// Mitsubishi GX Developer project: Пресс 40 (СКО)   PLC: FX3G

PROGRAM MAIN
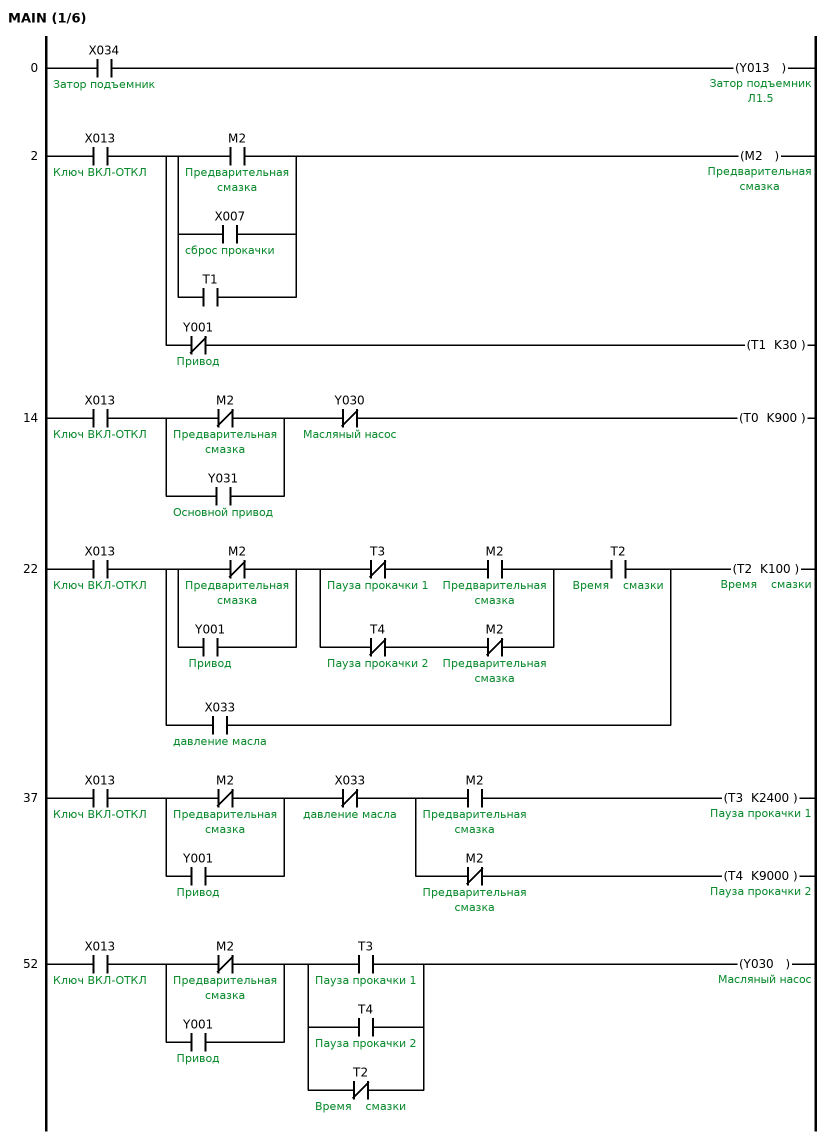
0     LD      X034  ; Затор подъемник
      OUT     Y013  ; Затор подъемник  Л1.5
2     LD      X013  ; Ключ ВКЛ-ОТКЛ
      MPS
      LD      M2  ; Предварительная смазка
      OR      X007  ; сброс прокачки
      OR      T1
      ANB
      OUT     M2  ; Предварительная смазка
      MPP
      ANI     Y001  ; Привод
      OUT     T1 K30
14    LD      X013  ; Ключ ВКЛ-ОТКЛ
      LDI     M2  ; Предварительная смазка
      OR      Y031  ; Основной привод
      ANB
      ANI     Y030  ; Масляный насос
      OUT     T0 K900
22    LD      X013  ; Ключ ВКЛ-ОТКЛ
      LDI     M2  ; Предварительная смазка
      OR      Y001  ; Привод
      LDI     T3  ; Пауза прокачки 1
      AND     M2  ; Предварительная смазка
      LDI     T4  ; Пауза прокачки 2
      ANI     M2  ; Предварительная смазка
      ORB
      ANB
      AND     T2  ; Время    смазки
      OR      X033  ; давление масла
      ANB
      OUT     T2 K100  ; Время    смазки
37    LD      X013  ; Ключ ВКЛ-ОТКЛ
      LDI     M2  ; Предварительная смазка
      OR      Y001  ; Привод
      ANB
      ANI     X033  ; давление масла
      MPS
      AND     M2  ; Предварительная смазка
      OUT     T3 K2400  ; Пауза прокачки 1
      MPP
      ANI     M2  ; Предварительная смазка
      OUT     T4 K9000  ; Пауза прокачки 2
52    LD      X013  ; Ключ ВКЛ-ОТКЛ
      LDI     M2  ; Предварительная смазка
      OR      Y001  ; Привод
      ANB
      LD      T3  ; Пауза прокачки 1
      OR      T4  ; Пауза прокачки 2
      ORI     T2  ; Время    смазки
      ANB
      OUT     Y030  ; Масляный насос
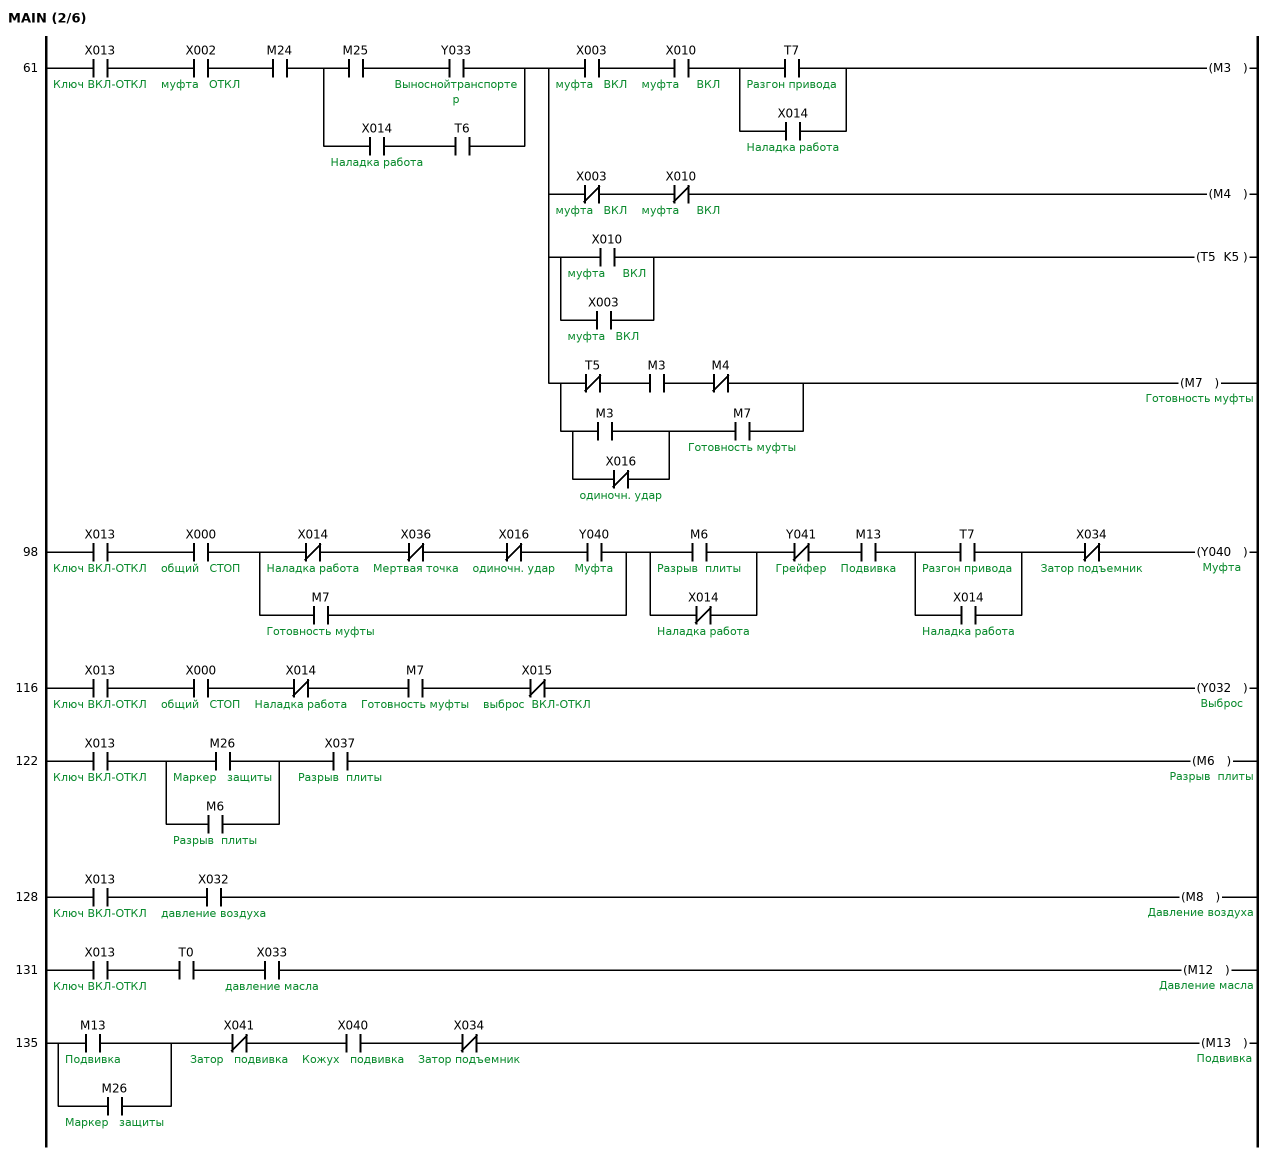
61    LD      X013  ; Ключ ВКЛ-ОТКЛ
      AND     X002  ; муфта   ОТКЛ
      AND     M24
      LD      M25
      AND     Y033  ; Выноснойтранспортер
      LD      X014  ; Наладка работа
      AND     T6
      ORB
      ANB
      MPS
      AND     X003  ; муфта   ВКЛ
      AND     X010  ; муфта     ВКЛ
      LD      T7  ; Разгон привода
      OR      X014  ; Наладка работа
      ANB
      OUT     M3
      MRD
      ANI     X003  ; муфта   ВКЛ
      ANI     X010  ; муфта     ВКЛ
      OUT     M4
      MRD
      LD      X010  ; муфта     ВКЛ
      OR      X003  ; муфта   ВКЛ
      ANB
      OUT     T5 K5
      MPP
      LDI     T5
      AND     M3
      ANI     M4
      LD      M3
      ORI     X016  ; одиночн. удар
      AND     M7  ; Готовность муфты
      ORB
      ANB
      OUT     M7  ; Готовность муфты
98    LD      X013  ; Ключ ВКЛ-ОТКЛ
      AND     X000  ; общий   СТОП
      LDI     X014  ; Наладка работа
      ANI     X036  ; Мертвая точка
      ANI     X016  ; одиночн. удар
      AND     Y040  ; Муфта
      OR      M7  ; Готовность муфты
      ANB
      LD      M6  ; Разрыв  плиты
      ORI     X014  ; Наладка работа
      ANB
      ANI     Y041  ; Грейфер
      AND     M13  ; Подвивка
      LD      T7  ; Разгон привода
      OR      X014  ; Наладка работа
      ANB
      ANI     X034  ; Затор подъемник
      OUT     Y040  ; Муфта
116   LD      X013  ; Ключ ВКЛ-ОТКЛ
      AND     X000  ; общий   СТОП
      ANI     X014  ; Наладка работа
      AND     M7  ; Готовность муфты
      ANI     X015  ; выброс  ВКЛ-ОТКЛ
      OUT     Y032  ; Выброс
122   LD      X013  ; Ключ ВКЛ-ОТКЛ
      LD      M26  ; Маркер   защиты
      OR      M6  ; Разрыв  плиты
      ANB
      AND     X037  ; Разрыв  плиты
      OUT     M6  ; Разрыв  плиты
128   LD      X013  ; Ключ ВКЛ-ОТКЛ
      AND     X032  ; давление воздуха
      OUT     M8  ; Давление воздуха
131   LD      X013  ; Ключ ВКЛ-ОТКЛ
      AND     T0
      AND     X033  ; давление масла
      OUT     M12  ; Давление масла
135   LD      M13  ; Подвивка
      OR      M26  ; Маркер   защиты
      ANI     X041  ; Затор   подвивка
      AND     X040  ; Кожух   подвивка
      ANI     X034  ; Затор подъемник
      OUT     M13  ; Подвивка
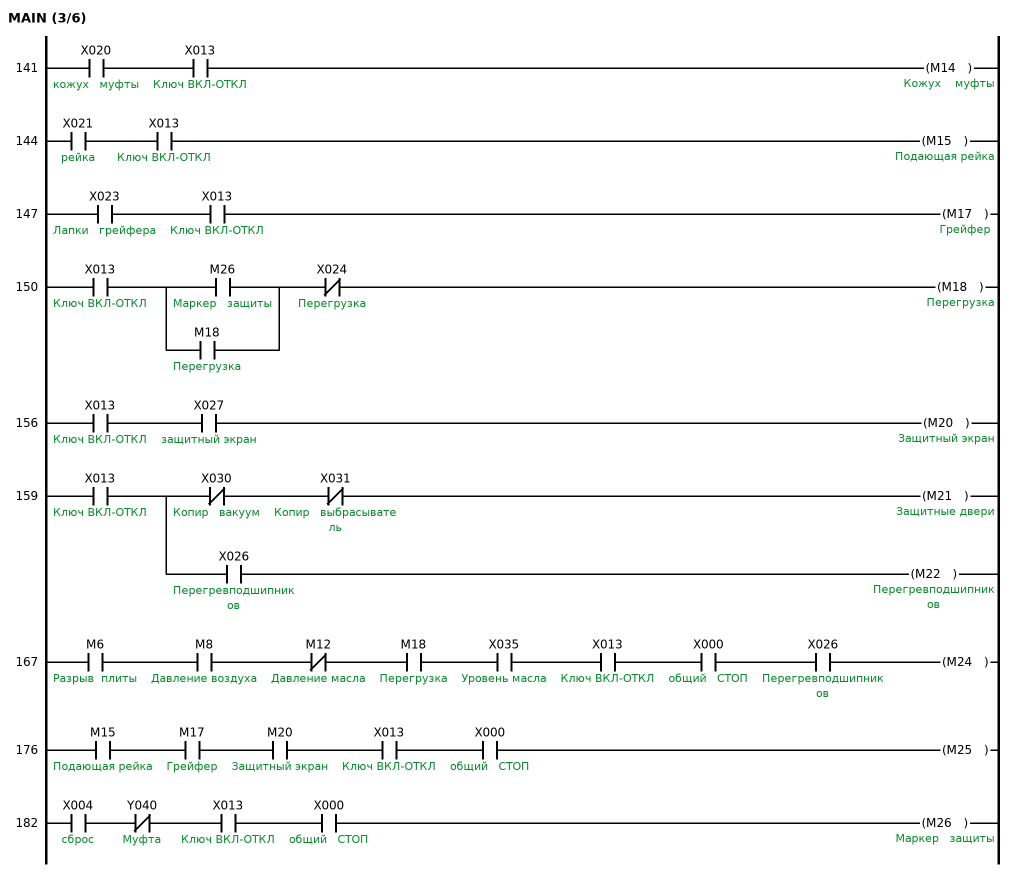
141   LD      X020  ; кожух   муфты
      AND     X013  ; Ключ ВКЛ-ОТКЛ
      OUT     M14  ; Кожух    муфты
144   LD      X021  ; рейка
      AND     X013  ; Ключ ВКЛ-ОТКЛ
      OUT     M15  ; Подающая рейка
147   LD      X023  ; Лапки   грейфера
      AND     X013  ; Ключ ВКЛ-ОТКЛ
      OUT     M17  ; Грейфер
150   LD      X013  ; Ключ ВКЛ-ОТКЛ
      LD      M26  ; Маркер   защиты
      OR      M18  ; Перегрузка
      ANB
      ANI     X024  ; Перегрузка
      OUT     M18  ; Перегрузка
156   LD      X013  ; Ключ ВКЛ-ОТКЛ
      AND     X027  ; защитный экран
      OUT     M20  ; Защитный экран
159   LD      X013  ; Ключ ВКЛ-ОТКЛ
      MPS
      ANI     X030  ; Копир   вакуум
      ANI     X031  ; Копир   выбрасыватель
      OUT     M21  ; Защитные двери
      MPP
      AND     X026  ; Перегревподшипников
      OUT     M22  ; Перегревподшипников
167   LD      M6  ; Разрыв  плиты
      AND     M8  ; Давление воздуха
      ANI     M12  ; Давление масла
      AND     M18  ; Перегрузка
      AND     X035  ; Уровень масла
      AND     X013  ; Ключ ВКЛ-ОТКЛ
      AND     X000  ; общий   СТОП
      AND     X026  ; Перегревподшипников
      OUT     M24
176   LD      M15  ; Подающая рейка
      AND     M17  ; Грейфер
      AND     M20  ; Защитный экран
      AND     X013  ; Ключ ВКЛ-ОТКЛ
      AND     X000  ; общий   СТОП
      OUT     M25
182   LD      X004  ; сброс
      ANI     Y040  ; Муфта
      AND     X013  ; Ключ ВКЛ-ОТКЛ
      AND     X000  ; общий   СТОП
      OUT     M26  ; Маркер   защиты
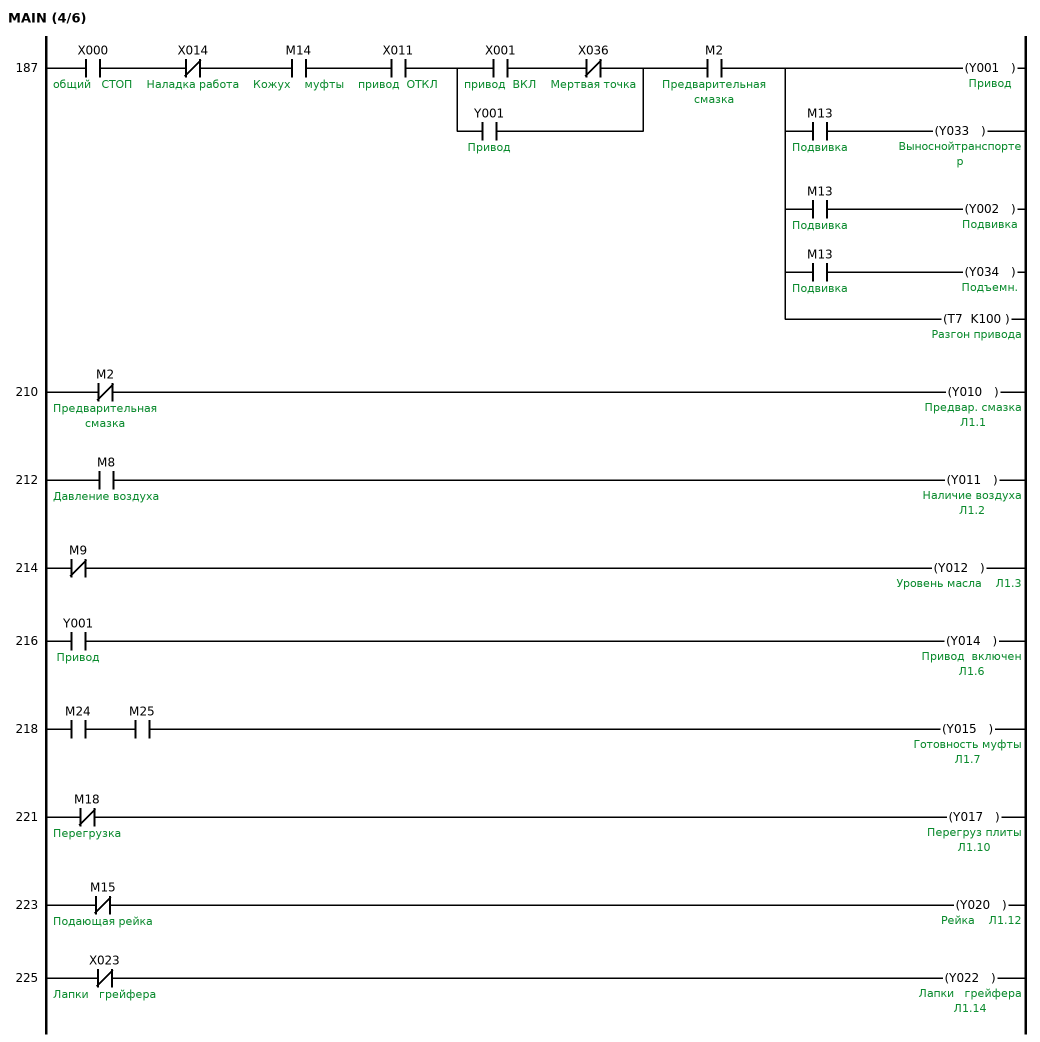
187   LD      X000  ; общий   СТОП
      ANI     X014  ; Наладка работа
      AND     M14  ; Кожух    муфты
      AND     X011  ; привод  ОТКЛ
      LD      X001  ; привод  ВКЛ
      ANI     X036  ; Мертвая точка
      OR      Y001  ; Привод
      ANB
      AND     M2  ; Предварительная смазка
      OUT     Y001  ; Привод
      MPS
      AND     M13  ; Подвивка
      OUT     Y033  ; Выноснойтранспортер
      MRD
      AND     M13  ; Подвивка
      OUT     Y002  ; Подвивка
      MRD
      AND     M13  ; Подвивка
      OUT     Y034  ; Подъемн.
      MPP
      OUT     T7 K100  ; Разгон привода
210   LDI     M2  ; Предварительная смазка
      OUT     Y010  ; Предвар. смазка   Л1.1
212   LD      M8  ; Давление воздуха
      OUT     Y011  ; Наличие воздуха  Л1.2
214   LDI     M9
      OUT     Y012  ; Уровень масла    Л1.3
216   LD      Y001  ; Привод
      OUT     Y014  ; Привод  включен  Л1.6
218   LD      M24
      AND     M25
      OUT     Y015  ; Готовность муфты  Л1.7
221   LDI     M18  ; Перегрузка
      OUT     Y017  ; Перегруз плиты   Л1.10
223   LDI     M15  ; Подающая рейка
      OUT     Y020  ; Рейка    Л1.12
225   LDI     X023  ; Лапки   грейфера
      OUT     Y022  ; Лапки   грейфера  Л1.14
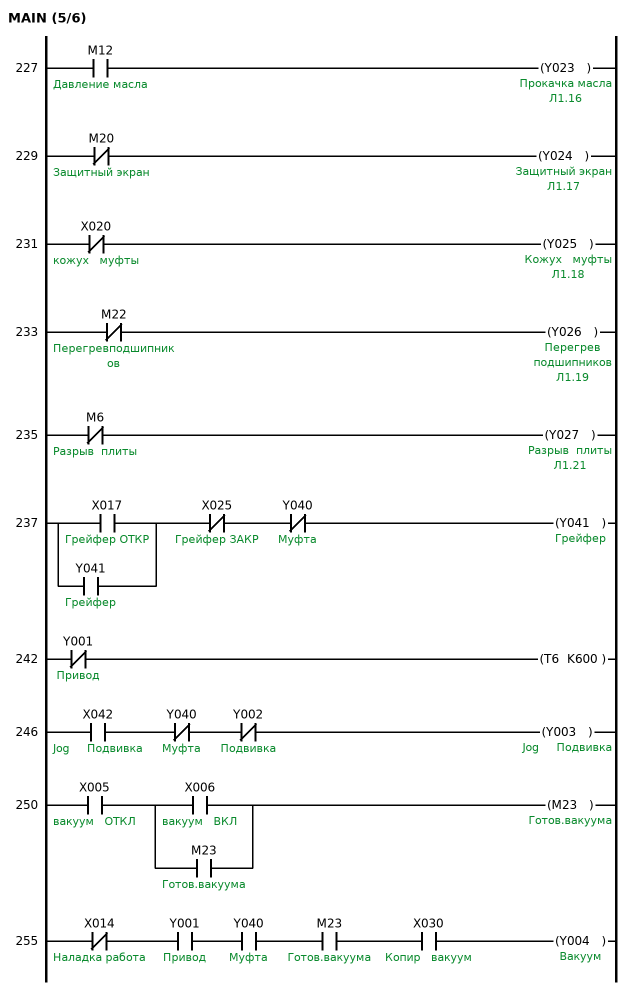
227   LD      M12  ; Давление масла
      OUT     Y023  ; Прокачка масла   Л1.16
229   LDI     M20  ; Защитный экран
      OUT     Y024  ; Защитный экран   Л1.17
231   LDI     X020  ; кожух   муфты
      OUT     Y025  ; Кожух   муфты   Л1.18
233   LDI     M22  ; Перегревподшипников
      OUT     Y026  ; Перегрев подшипников     Л1.19
235   LDI     M6  ; Разрыв  плиты
      OUT     Y027  ; Разрыв  плиты    Л1.21
237   LD      X017  ; Грейфер ОТКР
      OR      Y041  ; Грейфер
      ANI     X025  ; Грейфер ЗАКР
      ANI     Y040  ; Муфта
      OUT     Y041  ; Грейфер
242   LDI     Y001  ; Привод
      OUT     T6 K600
246   LD      X042  ; Jog     Подвивка
      ANI     Y040  ; Муфта
      ANI     Y002  ; Подвивка
      OUT     Y003  ; Jog     Подвивка
250   LD      X005  ; вакуум   ОТКЛ
      LD      X006  ; вакуум   ВКЛ
      OR      M23  ; Готов.вакуума
      ANB
      OUT     M23  ; Готов.вакуума
255   LDI     X014  ; Наладка работа
      AND     Y001  ; Привод
      AND     Y040  ; Муфта
      AND     M23  ; Готов.вакуума
      AND     X030  ; Копир   вакуум
      OUT     Y004  ; Вакуум
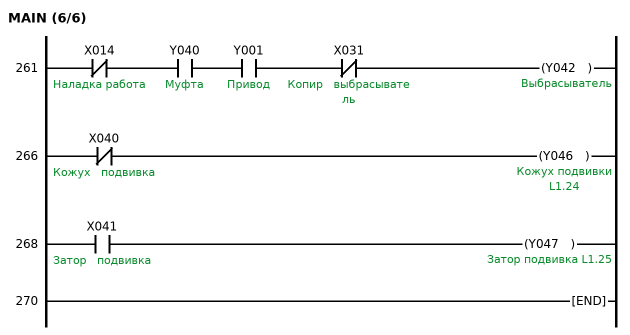
261   LDI     X014  ; Наладка работа
      AND     Y040  ; Муфта
      AND     Y001  ; Привод
      ANI     X031  ; Копир   выбрасыватель
      OUT     Y042  ; Выбрасыватель
266   LDI     X040  ; Кожух   подвивка
      OUT     Y046  ; Кожух подвивки L1.24
268   LD      X041  ; Затор   подвивка
      OUT     Y047  ; Затор подвивка L1.25
270   END
END_PROGRAM

// device comments not shown above
M1  ; Тепловая защита
M16  ; Выброс
M19  ; Перегрузка
X012  ; проверка ламп
X022  ; выбрасыватель
X043  ; Сдув    крышки
Y016  ; Выброс  открыт   Л1.8
Y021  ; Двойной лист
Y044  ; Подвивка
